{attribute 'qualified_only'}
{attribute 'strict'}
{attribute 'to_string'}
TYPE E_StartupState :
(
    STARTUP_IDLE:=0,
    STARTUP_CLEAR,
    STARTUP_RESET_FAULT,
    STARTUP_SHUTDOWN,
    STARTUP_SWITCH_ON,
    STARTUP_ENABLE_OP
);
END_TYPE

(* stored: Version 1.1.0.1
   DUT E_StartupState: Id {a438f9d9-85e4-4a52-b694-851762491b8a} *)
